PROGRAM X_Axis
VAR

END_VAR



TrucX();

METHOD nhap : BOOL
VAR_INPUT
END_VAR
// NETWORK 1

// NETWORK 2
END_METHOD

METHOD TrucX : BOOL
VAR_INPUT
END_VAR
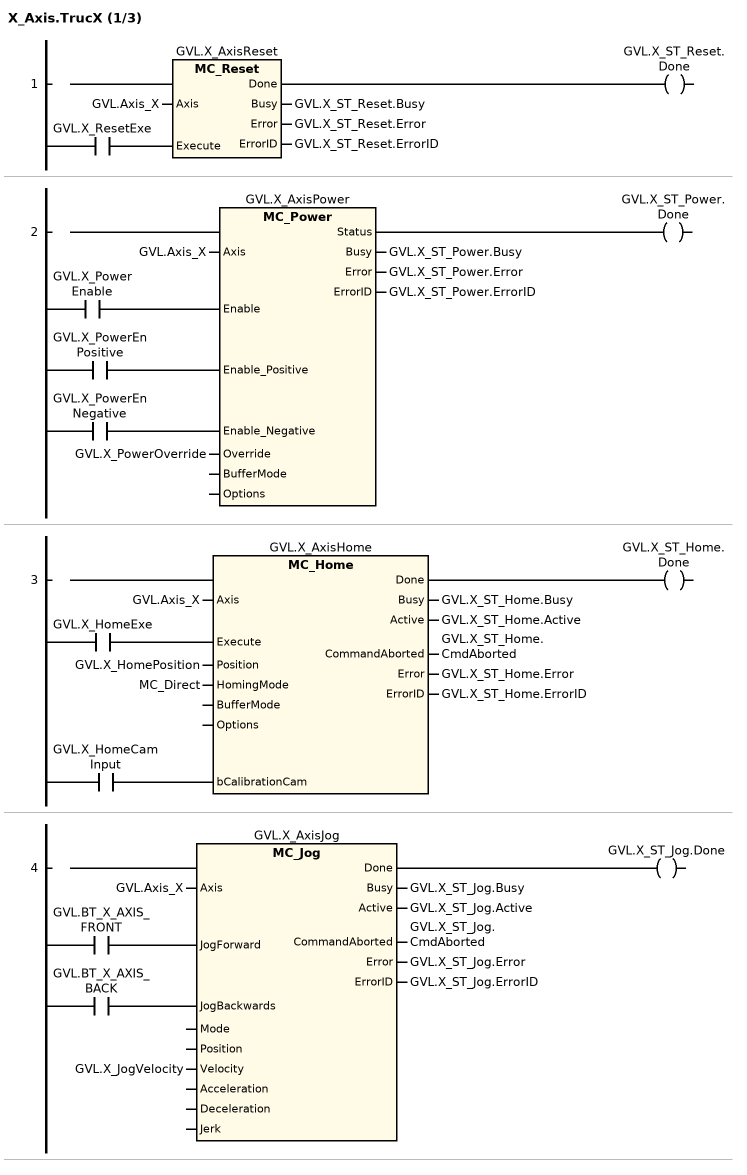
// NETWORK 1
GVL.X_AxisReset(
    Axis := GVL.Axis_X,
    Execute := GVL.X_ResetExe,
    Busy => GVL.X_ST_Reset.Busy,
    Error => GVL.X_ST_Reset.Error,
    ErrorID => GVL.X_ST_Reset.ErrorID); // MC_Reset
GVL.X_ST_Reset.Done := GVL.X_AxisReset.Done;

// NETWORK 2
GVL.X_AxisPower(
    Axis := GVL.Axis_X,
    Enable := GVL.X_PowerEnable,
    Enable_Positive := GVL.X_PowerEnPositive,
    Enable_Negative := GVL.X_PowerEnNegative,
    Override := GVL.X_PowerOverride,
    Busy => GVL.X_ST_Power.Busy,
    Error => GVL.X_ST_Power.Error,
    ErrorID => GVL.X_ST_Power.ErrorID); // MC_Power
GVL.X_ST_Power.Done := GVL.X_AxisPower.Status;

// NETWORK 3
GVL.X_AxisHome(
    Axis := GVL.Axis_X,
    Execute := GVL.X_HomeExe,
    Position := GVL.X_HomePosition,
    HomingMode := MC_Direct,
    bCalibrationCam := GVL.X_HomeCamInput,
    Busy => GVL.X_ST_Home.Busy,
    Active => GVL.X_ST_Home.Active,
    CommandAborted => GVL.X_ST_Home.CmdAborted,
    Error => GVL.X_ST_Home.Error,
    ErrorID => GVL.X_ST_Home.ErrorID); // MC_Home
GVL.X_ST_Home.Done := GVL.X_AxisHome.Done;

// NETWORK 4
GVL.X_AxisJog(
    Axis := GVL.Axis_X,
    JogForward := GVL.BT_X_AXIS_FRONT,
    JogBackwards := GVL.BT_X_AXIS_BACK,
    Velocity := GVL.X_JogVelocity,
    Busy => GVL.X_ST_Jog.Busy,
    Active => GVL.X_ST_Jog.Active,
    CommandAborted => GVL.X_ST_Jog.CmdAborted,
    Error => GVL.X_ST_Jog.Error,
    ErrorID => GVL.X_ST_Jog.ErrorID); // MC_Jog
GVL.X_ST_Jog.Done := GVL.X_AxisJog.Done;

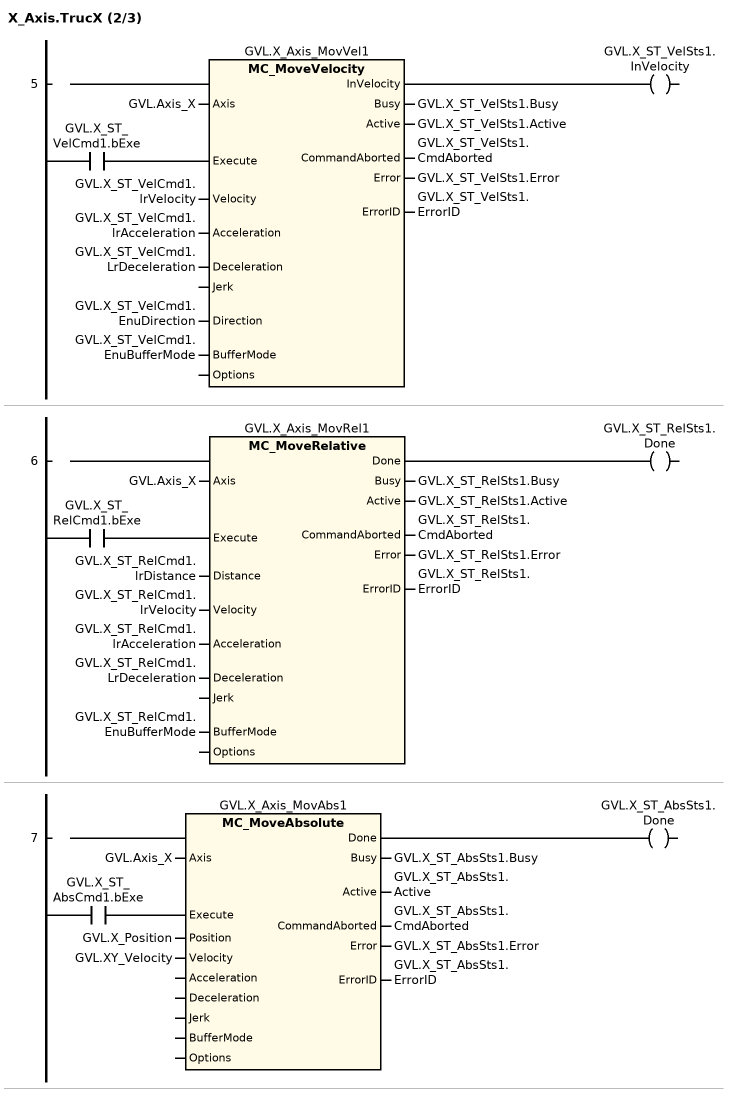
// NETWORK 5
GVL.X_Axis_MovVel1(
    Axis := GVL.Axis_X,
    Execute := GVL.X_ST_VelCmd1.bExe,
    Velocity := GVL.X_ST_VelCmd1.lrVelocity,
    Acceleration := GVL.X_ST_VelCmd1.lrAcceleration,
    Deceleration := GVL.X_ST_VelCmd1.LrDeceleration,
    Direction := GVL.X_ST_VelCmd1.EnuDirection,
    BufferMode := GVL.X_ST_VelCmd1.EnuBufferMode,
    Busy => GVL.X_ST_VelSts1.Busy,
    Active => GVL.X_ST_VelSts1.Active,
    CommandAborted => GVL.X_ST_VelSts1.CmdAborted,
    Error => GVL.X_ST_VelSts1.Error,
    ErrorID => GVL.X_ST_VelSts1.ErrorID); // MC_MoveVelocity
GVL.X_ST_VelSts1.InVelocity := GVL.X_Axis_MovVel1.InVelocity;

// NETWORK 6
GVL.X_Axis_MovRel1(
    Axis := GVL.Axis_X,
    Execute := GVL.X_ST_RelCmd1.bExe,
    Distance := GVL.X_ST_RelCmd1.lrDistance,
    Velocity := GVL.X_ST_RelCmd1.lrVelocity,
    Acceleration := GVL.X_ST_RelCmd1.lrAcceleration,
    Deceleration := GVL.X_ST_RelCmd1.LrDeceleration,
    BufferMode := GVL.X_ST_RelCmd1.EnuBufferMode,
    Busy => GVL.X_ST_RelSts1.Busy,
    Active => GVL.X_ST_RelSts1.Active,
    CommandAborted => GVL.X_ST_RelSts1.CmdAborted,
    Error => GVL.X_ST_RelSts1.Error,
    ErrorID => GVL.X_ST_RelSts1.ErrorID); // MC_MoveRelative
GVL.X_ST_RelSts1.Done := GVL.X_Axis_MovRel1.Done;

// NETWORK 7
GVL.X_Axis_MovAbs1(
    Axis := GVL.Axis_X,
    Execute := GVL.X_ST_AbsCmd1.bExe,
    Position := GVL.X_Position,
    Velocity := GVL.XY_Velocity,
    Busy => GVL.X_ST_AbsSts1.Busy,
    Active => GVL.X_ST_AbsSts1.Active,
    CommandAborted => GVL.X_ST_AbsSts1.CmdAborted,
    Error => GVL.X_ST_AbsSts1.Error,
    ErrorID => GVL.X_ST_AbsSts1.ErrorID); // MC_MoveAbsolute
GVL.X_ST_AbsSts1.Done := GVL.X_Axis_MovAbs1.Done;

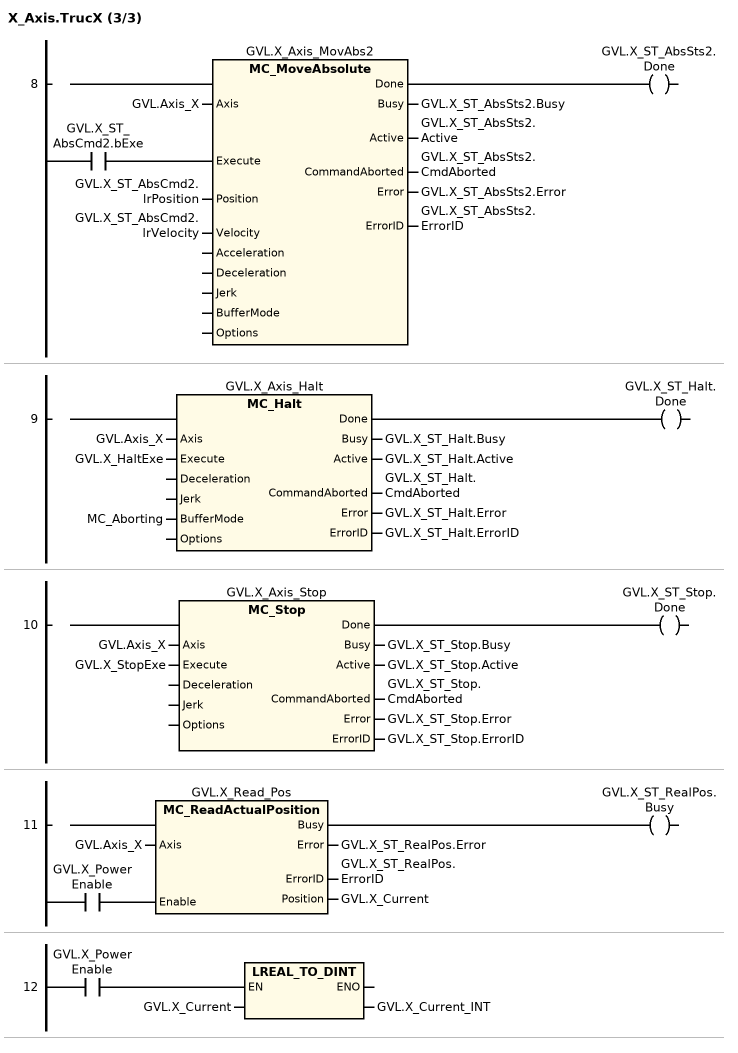
// NETWORK 8
GVL.X_Axis_MovAbs2(
    Axis := GVL.Axis_X,
    Execute := GVL.X_ST_AbsCmd2.bExe,
    Position := GVL.X_ST_AbsCmd2.lrPosition,
    Velocity := GVL.X_ST_AbsCmd2.lrVelocity,
    Busy => GVL.X_ST_AbsSts2.Busy,
    Active => GVL.X_ST_AbsSts2.Active,
    CommandAborted => GVL.X_ST_AbsSts2.CmdAborted,
    Error => GVL.X_ST_AbsSts2.Error,
    ErrorID => GVL.X_ST_AbsSts2.ErrorID); // MC_MoveAbsolute
GVL.X_ST_AbsSts2.Done := GVL.X_Axis_MovAbs2.Done;

// NETWORK 9
GVL.X_Axis_Halt(
    Axis := GVL.Axis_X,
    Execute := GVL.X_HaltExe,
    BufferMode := MC_Aborting,
    Busy => GVL.X_ST_Halt.Busy,
    Active => GVL.X_ST_Halt.Active,
    CommandAborted => GVL.X_ST_Halt.CmdAborted,
    Error => GVL.X_ST_Halt.Error,
    ErrorID => GVL.X_ST_Halt.ErrorID); // MC_Halt
GVL.X_ST_Halt.Done := GVL.X_Axis_Halt.Done;

// NETWORK 10
GVL.X_Axis_Stop(
    Axis := GVL.Axis_X,
    Execute := GVL.X_StopExe,
    Busy => GVL.X_ST_Stop.Busy,
    Active => GVL.X_ST_Stop.Active,
    CommandAborted => GVL.X_ST_Stop.CmdAborted,
    Error => GVL.X_ST_Stop.Error,
    ErrorID => GVL.X_ST_Stop.ErrorID); // MC_Stop
GVL.X_ST_Stop.Done := GVL.X_Axis_Stop.Done;

// NETWORK 11
GVL.X_Read_Pos(
    Axis := GVL.Axis_X,
    Enable := GVL.X_PowerEnable,
    Busy => GVL.X_ST_RealPos.Busy,
    Error => GVL.X_ST_RealPos.Error,
    ErrorID => GVL.X_ST_RealPos.ErrorID,
    Position => GVL.X_Current); // MC_ReadActualPosition

// NETWORK 12
IF GVL.X_PowerEnable THEN GVL.X_Current_INT := LREAL_TO_DINT(GVL.X_Current); END_IF
END_METHOD

END_PROGRAM

(* stored: Version 1.1.0.1, ProductVersion 3.1.4024.13
   POU X_Axis: Id {792fa090-3240-4073-a837-286c62690c4a}, SpecialFunc None
   Method nhap: Id {e4b48dd9-43ef-4984-a788-ceaef17b43a4}
   Method TrucX: Id {7dede1ce-9040-47d1-b228-bfc1f8b41fbc} *)
